Fanuc KAREL source: IO0196.KL

-- PROVISIONAL review KL for V940-1; original PC SHA256 3df6f3ff4bd4af79dc073b603663b48f2db8f9c164bac20e4ac04ce828026326
-- Incomplete behavior may be omitted. Consult companion uncertainty JSON. Do not deploy.
PROGRAM IO0196
%NOLOCKGROUP
-- UNRESOLVED_LOCAL_POOL 5 cells at code offset 13; source declarations unknown
-- DIRECT_LOCAL_WORD_ACCESS alone does not prove INTEGER, REAL, or BOOLEAN
BEGIN
  -- V9_EXPOSED_INDEXED_TABLE_HINT layout=0002_ascii; 1 counted words exposed once; source arms/runtime held
  -- V9_INDEXED_0002_HINT 1 indexed wire operands; static native loader address link; source ownership held
  -- UNRESOLVED_PC offsets 0-18; opcodes 2B,2C,7B
  -- UNRESOLVED_PC offsets 23-30; opcodes 9D,23
  -- UNRESOLVED_PC offsets 35-49; opcodes 2E,22,9D,33,35
  -- UNRESOLVED_PC offsets 54-61; opcodes 9D,23
  -- UNRESOLVED_PC offsets 66-77; opcodes 2E,23
  -- UNRESOLVED_PC offsets 82-108; opcodes 27,27,9D,22,27,9D,31,7E,4A
  -- UNRESOLVED_PC offsets 113-130; opcodes 22,32,34,9C,71,79
  -- UNRESOLVED_PC offsets 135-149; opcodes 21,9D,52,23
  -- UNRESOLVED_PC offsets 159-163; opcodes 7F
  -- UNRESOLVED_PC offsets 168-172; opcodes 27,AA
  -- UNRESOLVED_PC offsets 177-181; opcodes 7F
END IO0196
